Yaskawa INFORM job: OK_R2_O48(150,-90)AWOK.JBI

/JOB
//NAME OK_R2_O48(150,-90)AWOK
///FOLDERNAME X4
//POS
///NPOS 93,93,93,5,0,0
///TOOL 0
///POSTYPE PULSE
///PULSE
C00000=7128,-162535,-102538,14833,-6408,52690
C00001=-104208,-118770,-74284,45981,33291,-26248
C00002=-127942,-89719,-58931,35307,42397,-46473
C00003=-123853,-84206,-54688,32906,40963,-44702
C00004=-120909,-81305,-52666,30982,40073,-43338
C00005=-120909,-80580,-51168,31322,39602,-43537
C00006=-120933,-81321,-52095,31218,39773,-43479
C00007=-120933,-81321,-52095,31218,39773,-43479
C00008=-118429,-81278,-52077,29602,38889,-42349
C00009=-119470,-83685,-55381,29802,39949,-42541
C00010=-120965,-86018,-57149,30812,40385,-43243
C00011=-124957,-91780,-61448,33373,41616,-45066
C00012=-119941,-104378,-75649,664,44366,-1357
C00013=-114575,-89440,-58348,-34911,41926,46281
C00014=-118628,-83889,-54076,-32484,40527,44503
C00015=-120150,-81634,-52317,-31517,40024,43814
C00016=-120153,-79883,-49949,-31862,39544,44015
C00017=-120152,-80596,-50915,-31720,39740,43932
C00018=-120152,-80596,-50915,-31720,39740,43932
C00019=-122990,-80556,-50898,-29906,38725,42654
C00020=-120487,-84798,-55273,-31191,40066,43596
C00021=-118937,-87092,-57018,-32198,40551,44309
C00022=-106067,-91307,-60720,-38685,45933,49349
C00023=-98484,-126815,-102076,-39276,55586,49844
C00024=-116041,-74769,-88862,-24389,64621,38504
C00025=-110869,-91165,-78577,-23331,92195,43854
C00026=-124249,-90532,-74394,-23419,86323,40078
C00027=-124579,-90250,-73658,-23419,85946,40029
C00028=-124579,-89705,-72166,-23424,85359,40146
C00029=-124579,-90004,-72979,-23418,85679,40084
C00030=-124579,-90004,-72979,-23418,85679,40084
C00031=-127139,-89747,-72875,-23368,85013,39271
C00032=-124513,-91644,-75080,-23411,86111,40023
C00033=-122390,-96046,-81338,-23429,88175,40400
C00034=-118210,-97090,-84712,-23461,90782,41427
C00035=-128682,-92973,-79431,23550,91181,-43199
C00036=-121322,-93591,-77129,23613,87481,-41217
C00037=-119783,-92676,-74656,23621,86073,-40929
C00038=-119783,-92003,-72902,23631,85399,-41062
C00039=-119783,-92315,-73705,23625,85706,-41001
C00040=-117303,-92210,-73665,23606,85023,-40222
C00041=-119476,-92309,-74377,23618,86001,-40830
C00042=-123453,-92705,-79015,23614,89575,-41589
C00043=-126833,-58246,-59490,24431,96195,-34985
C00044=-121064,-58502,-56942,24348,92946,-33515
C00045=-122349,-90639,-72271,24283,86838,-35236
C00046=-120613,-91235,-73784,24290,86900,-34580
C00047=-121081,-75684,-65541,24266,89714,-34181
C00048=-121026,-92775,-72870,24282,85789,-34961
C00049=-121053,-101624,-76099,24352,83453,-35450
C00050=-121053,-101774,-76152,24354,83412,-35459
C00051=-121214,-86270,-68515,24620,98676,-32382
C00052=-121315,-89830,-69273,24565,98526,-32452
C00053=-128764,-80026,-69192,23683,105275,-33882
C00054=-134806,-66986,-70278,23625,104239,-34458
C00055=-107842,-77648,-85221,-23587,98114,40069
C00056=-119915,-70001,-63560,-27444,90659,45675
C00057=-122863,-62004,-57325,-27391,89936,44725
C00058=-125343,-108335,-78841,-26517,77272,26818
C00059=-123289,-107584,-77287,-26635,77411,27568
C00060=-123156,-76901,-64612,-27381,87009,45299
C00061=-123624,-94441,-71953,-27500,82842,46100
C00062=-123937,-107499,-76607,-27734,79312,46822
C00063=-123895,-107588,-76637,-27736,79301,46841
C00064=-124111,-102845,-74409,-27467,87071,44933
C00065=-123700,-99391,-71448,-27908,92704,43616
C00066=-123818,-102887,-72152,-27884,91453,43871
C00067=-113172,-80591,-67120,-26641,104065,45143
C00068=-103355,-56663,-86718,-43856,106110,10768
C00069=-95822,-140722,-117880,-57553,87470,-6427
C00070=-59504,-196684,-108230,-85963,76535,-42215
C00071=-126651,-173103,-98619,-107590,31890,-42335
C00072=-132485,-146292,-95297,-89338,25934,-52354
C00073=-127502,-141387,-93667,-80295,34491,-61924
C00074=-120359,-173692,-85938,-119295,41762,-37936
C00075=-112237,-170659,-84465,-112953,45862,-39581
C00076=-127507,-141456,-93682,-80333,34482,-61904
C00077=-127989,-162289,-111384,-72485,35866,-66585
C00078=-127720,-186855,-131843,-64092,39200,-71745
C00079=-127563,-185307,-132809,-61202,40726,-73506
C00080=-141972,-165441,-94982,-91935,28434,-22119
C00081=-120670,-166785,-110893,11236,47417,-7793
C00082=-120378,-170313,-84464,114311,39014,41261
C00083=-118671,-173407,-93959,109670,36018,44646
C00084=-117490,-116273,-97513,47995,52698,87558
C00085=-128335,-170190,-84462,108879,43427,42364
C00086=-120365,-173150,-86026,114896,39194,40925
C00087=-117457,-117591,-97936,48216,52395,87392
C00088=-108592,-156504,-118933,44933,39836,84216
C00089=-108710,-192099,-136125,56896,33409,77883
C00090=-110038,-135908,-122263,39784,48159,87867
C00091=-30894,-171068,-100229,56651,5883,46742
C00092=7128,-162535,-102538,14833,-6408,52690
BC00000=199595,668284,1075175
BC00001=291872,675689,1075175
BC00002=333462,679027,1075175
BC00003=333462,679027,1075175
BC00004=333462,679027,1075175
BC00005=333462,679027,1075175
BC00006=333462,679027,1075175
BC00007=333462,679027,1075175
BC00008=333462,679027,1075175
BC00009=333462,679027,1075175
BC00010=333462,679027,1075175
BC00011=333462,679027,1075175
BC00012=223299,677892,1075175
BC00013=102985,676652,1075175
BC00014=102985,676652,1075175
BC00015=102985,676652,1075175
BC00016=102985,676652,1075175
BC00017=102985,676652,1075175
BC00018=102985,676652,1075175
BC00019=102985,676652,1075175
BC00020=102985,676652,1075175
BC00021=102985,676652,1075175
BC00022=102985,676652,1075175
BC00023=102985,676652,1075175
BC00024=102985,676652,1075175
BC00025=115373,806609,1075175
BC00026=115373,806609,1075175
BC00027=115373,806609,1075175
BC00028=115373,806609,1075175
BC00029=115373,806609,1075175
BC00030=115373,806609,1075175
BC00031=115373,806609,1075175
BC00032=115373,806609,1075175
BC00033=115373,806609,1075175
BC00034=115373,806609,1075175
BC00035=324585,809621,1075175
BC00036=324585,809621,1075175
BC00037=324585,809621,1075175
BC00038=324585,809621,1075175
BC00039=324585,809621,1075175
BC00040=324585,809621,1075175
BC00041=324585,809621,1075175
BC00042=324585,809621,1075175
BC00043=328987,784971,1075168
BC00044=328987,784971,1075168
BC00045=328987,784969,1075175
BC00046=328987,784969,1075175
BC00047=328987,784971,1075168
BC00048=328987,784971,1075168
BC00049=328987,784971,1075168
BC00050=328987,784971,1075168
BC00051=328987,784971,1075168
BC00052=328987,784971,1075168
BC00053=328987,784971,1075168
BC00054=328987,784971,1075168
BC00055=116574,792346,1075173
BC00056=116574,792346,1075173
BC00057=116574,792346,1075173
BC00058=116574,792346,1075175
BC00059=116574,792346,1075175
BC00060=116574,792346,1075173
BC00061=116574,792346,1075173
BC00062=116574,792346,1075173
BC00063=116574,792346,1075173
BC00064=116574,792346,1075173
BC00065=116575,792346,1075173
BC00066=116575,792346,1075173
BC00067=116574,792346,1075173
BC00068=116574,737436,1075175
BC00069=122857,733121,993715
BC00070=135433,724483,830653
BC00071=135432,724483,830653
BC00072=135433,724483,830653
BC00073=135433,724483,830653
BC00074=127658,730199,812564
BC00075=127658,730199,812564
BC00076=135433,724483,830653
BC00077=135433,724483,830653
BC00078=135433,724483,830653
BC00079=135433,724483,830653
BC00080=160615,710357,862138
BC00081=210523,682360,924538
BC00082=303867,722052,847743
BC00083=303867,722052,847743
BC00084=303867,722052,847743
BC00085=311621,727375,828139
BC00086=311621,727375,828139
BC00087=303867,722052,847743
BC00088=303867,722052,847743
BC00089=303867,722052,847743
BC00090=276888,676778,849704
BC00091=235848,686978,996103
BC00092=199595,668284,1075175
EC00000=1330261,-556475
EC00001=1330261,-556475
EC00002=1330261,-556475
EC00003=1330261,-556475
EC00004=1330261,-556475
EC00005=1330261,-556475
EC00006=1330261,-556475
EC00007=1330261,-556475
EC00008=1330261,-556475
EC00009=1330261,-556475
EC00010=1330261,-556475
EC00011=1330261,-556475
EC00012=1330261,-556475
EC00013=1330261,-556475
EC00014=1330261,-556475
EC00015=1330261,-556475
EC00016=1330261,-556475
EC00017=1330261,-556475
EC00018=1330261,-556475
EC00019=1330261,-556475
EC00020=1330261,-556475
EC00021=1330261,-556475
EC00022=1330261,-556475
EC00023=1330261,-556475
EC00024=1330261,-556475
EC00025=1330261,-556475
EC00026=1330261,-556475
EC00027=1330261,-556475
EC00028=1330261,-556475
EC00029=1330261,-556475
EC00030=1330261,-556475
EC00031=1330261,-556475
EC00032=1330261,-556475
EC00033=1330261,-556475
EC00034=1330261,-556475
EC00035=1330261,-556475
EC00036=1330261,-556475
EC00037=1330261,-556475
EC00038=1330261,-556475
EC00039=1330261,-556475
EC00040=1330261,-556475
EC00041=1330261,-556475
EC00042=1330261,-556475
EC00043=1330260,-556475
EC00044=1330260,-556475
EC00045=1330261,-556475
EC00046=1330261,-556475
EC00047=1330260,-556475
EC00048=1330260,-556475
EC00049=1330260,-556475
EC00050=1330260,-556475
EC00051=1330260,-556475
EC00052=1330260,-556475
EC00053=1330260,-556475
EC00054=1330260,-556475
EC00055=1330261,-556475
EC00056=1330261,-556475
EC00057=1330261,-556475
EC00058=1330261,-556475
EC00059=1330261,-556475
EC00060=1330261,-556475
EC00061=1330261,-556475
EC00062=1330261,-556475
EC00063=1330261,-556475
EC00064=1330261,-556475
EC00065=1330261,-556475
EC00066=1330261,-556475
EC00067=1330261,-556475
EC00068=1330261,-556475
EC00069=1330261,-556475
EC00070=1330261,-556475
EC00071=1330261,-556475
EC00072=1330261,-556475
EC00073=1330261,-556475
EC00074=1330261,-556475
EC00075=1330261,-556475
EC00076=1330261,-556475
EC00077=1276882,-556475
EC00078=1207176,-556475
EC00079=1207176,-556475
EC00080=1330261,-556475
EC00081=1330261,-556475
EC00082=1330261,-556475
EC00083=1330261,-556475
EC00084=1330261,-556475
EC00085=1330261,-556475
EC00086=1330261,-556475
EC00087=1330261,-556475
EC00088=1270757,-556475
EC00089=1191966,-556475
EC00090=1191966,-556475
EC00091=1330261,-556475
EC00092=1330261,-556475
///POSTYPE BASE
///RECTAN
///RCONF 0,0,0,0,0,0,0,0,0,0,0,0,0,0,0,0,0,0,0,0,0,0,0,0
P00006=0.222,-3.123,-1.508,0.0000,0.0000,0.0000
P00021=-0.225,-6.128,-0.405,0.0000,0.0000,0.0000
P00022=0.222,-3.123,-1.508,0.0000,0.0000,0.0000
P00031=1.853,-0.001,-1.549,0.0000,0.0000,0.0000
P00032=1.957,0.503,-7.217,0.0000,0.0000,0.0000
//INST
///DATE 2025/02/06 10:35
///ATTR SC,RW
///GROUP1 RB1,BS1
///GROUP2 ST1
///LVARS 0,0,0,0,0,100,0,0
NOP
'OK_r2_O48(150,-90)
'Path S1531
MOVJ C00000 BC00000 VJ=100.00  +MOVJ EC00000 VJ=50.00
SFTOF3D
MOVJ C00001 BC00001 VJ=100.00  +MOVJ EC00001 VJ=50.00
MOVJ C00002 BC00002 VJ=100.00  +MOVJ EC00002 VJ=100.00
MOVL C00003 BC00003 V=400.0  +MOVJ EC00003 VJ=100.00
SMOVL C00004 BC00004 V=100.0  +MOVJ EC00004
SREFP 3 C00005 BC00005  +REFP EC00005
CALL JOB:SEARCH-R1-S13D
SET P021 P006
SFTON3D P021
SMOVL C00006 BC00006 V=100.0  +MOVJ EC00006
SMOVL C00007 BC00007 V=100.0  +MOVJ EC00007
SREFP 3 C00008 BC00008  +REFP EC00008
CALL JOB:SEARCH-R1-S13D
SET P021 P006
SFTON3D P021
SMOVL C00009 BC00009 V=100.0  +MOVJ EC00009
MOVL C00010 BC00010 V=400.0  +MOVJ EC00010 VJ=100.00
MOVL C00011 BC00011 V=1000.0  +MOVJ EC00011 VJ=100.00
'Path S1532
SFTOF3D
MOVJ C00012 BC00012 VJ=100.00  +MOVJ EC00012 VJ=10.00
MOVJ C00013 BC00013 VJ=100.00  +MOVJ EC00013 VJ=100.00
MOVL C00014 BC00014 V=333.3  +MOVJ EC00014 VJ=100.00
SMOVL C00015 BC00015 V=100.0  +MOVJ EC00015
SREFP 3 C00016 BC00016  +REFP EC00016
CALL JOB:SEARCH-R1-S13D
SET P022 P006
SFTON3D P022
SMOVL C00017 BC00017 V=100.0  +MOVJ EC00017
SMOVL C00018 BC00018 V=100.0  +MOVJ EC00018
SREFP 3 C00019 BC00019  +REFP EC00019
CALL JOB:SEARCH-R1-S13D
SET P022 P006
SFTON3D P022
SMOVL C00020 BC00020 V=100.0  +MOVJ EC00020
MOVL C00021 BC00021 V=400.0  +MOVJ EC00021 VJ=100.00
MOVL C00022 BC00022 V=1000.0  +MOVJ EC00022 VJ=100.00
MOVJ C00023 BC00023 VJ=100.00  +MOVJ EC00023 VJ=50.00
MOVJ C00024 BC00024 VJ=100.00  +MOVJ EC00024 VJ=100.00
'Path S1235
SFTOF3D
MOVJ C00025 BC00025 VJ=100.00  +MOVJ EC00025 VJ=100.00
MOVL C00026 BC00026 V=400.0  +MOVJ EC00026 VJ=100.00
SMOVL C00027 BC00027 V=100.0  +MOVJ EC00027
SREFP 3 C00028 BC00028  +REFP EC00028
CALL JOB:SEARCH-R1-S13D
SET P032 P006
SFTON3D P032
SMOVL C00029 BC00029 V=100.0  +MOVJ EC00029
SMOVL C00030 BC00030 V=100.0  +MOVJ EC00030
SREFP 3 C00031 BC00031  +REFP EC00031
CALL JOB:SEARCH-R1-S13D
SET P032 P006
SFTON3D P032
SMOVL C00032 BC00032 V=100.0  +MOVJ EC00032
MOVL C00033 BC00033 V=400.0  +MOVJ EC00033 VJ=100.00
MOVL C00034 BC00034 V=1000.0  +MOVJ EC00034 VJ=100.00
'Path S1204
SFTOF3D
MOVJ C00035 BC00035 VJ=100.00  +MOVJ EC00035 VJ=100.00
MOVL C00036 BC00036 V=400.0  +MOVJ EC00036 VJ=100.00
SMOVL C00037 BC00037 V=100.0  +MOVJ EC00037
SREFP 3 C00038 BC00038  +REFP EC00038
CALL JOB:SEARCH-R1-S13D
SET P031 P006
SFTON3D P031
SMOVL C00039 BC00039 V=100.0  +MOVJ EC00039
SREFP 3 C00040 BC00040  +REFP EC00040
CALL JOB:SEARCH-R1-S13D
SET P031 P006
SFTON3D P031
SMOVL C00041 BC00041 V=100.0  +MOVJ EC00041
MOVL C00042 BC00042 V=400.0  +MOVJ EC00042 VJ=100.00
SFTOF3D
'Path W341
SFTOF3D
SFTON3D P031
SMOVL C00043 BC00043 V=400.0  +MOVJ EC00043
SMOVL C00044 BC00044 V=400.0 PL=0  +MOVJ EC00044
SREFP 1 C00045 BC00045  +REFP EC00045
SREFP 2 C00046 BC00046  +REFP EC00046
MACRO1 MJ#(0) ARGF21
ARCON
SWVON WEV#(101)
SMOVL C00047 BC00047 V=8.3  +MOVJ EC00047
SMOVL C00048 BC00048 V=8.3  +MOVJ EC00048
SMOVL C00049 BC00049 V=8.3  +MOVJ EC00049
SMOVC C00050 BC00050 V=8.3  +MOVJ EC00050
SMOVC C00051 BC00051 V=8.3  +MOVJ EC00051
SMOVC C00052 BC00052 V=8.3  +MOVJ EC00052
ARCOF
SFTOF3D
SWVOF
SMOVL C00053 BC00053 V=250.0  +MOVJ EC00053
MOVJ C00054 BC00054 VJ=100.00  +MOVJ EC00054 VJ=100.00
MOVJ C00055 BC00055 VJ=100.00  +MOVJ EC00055 VJ=100.00
SFTOF3D
'Path W2042
SFTOF3D
SFTON3D P032
SMOVL C00056 BC00056 V=400.0  +MOVJ EC00056
SMOVL C00057 BC00057 V=166.7 PL=0  +MOVJ EC00057
SREFP 1 C00058 BC00058  +REFP EC00058
SREFP 2 C00059 BC00059  +REFP EC00059
ARCON
SWVON WEV#(101)
SMOVL C00060 BC00060 V=8.3  +MOVJ EC00060
SMOVL C00061 BC00061 V=8.3  +MOVJ EC00061
SMOVL C00062 BC00062 V=8.3  +MOVJ EC00062
SMOVC C00063 BC00063 V=8.3  +MOVJ EC00063
SMOVC C00064 BC00064 V=8.3  +MOVJ EC00064
SMOVC C00065 BC00065 V=10.0  +MOVJ EC00065
SMOVC C00066 BC00066 V=10.0  +MOVJ EC00066
ARCOF
SWVOF
SMOVL C00067 BC00067 V=400.0  +MOVJ EC00067
SFTOF3D
MOVJ C00068 BC00068 VJ=100.00  +MOVJ EC00068 VJ=100.00
MOVJ C00069 BC00069 VJ=100.00  +MOVJ EC00069 VJ=50.00
MOVJ C00070 BC00070 VJ=100.00  +MOVJ EC00070 VJ=100.00
SFTOF3D
'Path W1533
SFTOF3D
SFTON3D P022
MOVJ C00071 BC00071 VJ=100.00  +MOVJ EC00071 VJ=50.00
SMOVL C00072 BC00072 V=400.0  +MOVJ EC00072
SMOVL C00073 BC00073 V=133.3 PL=0  +MOVJ EC00073
SREFP 1 C00074 BC00074  +REFP EC00074
SREFP 2 C00075 BC00075  +REFP EC00075
ARCON
SWVON WEV#(101)
SMOVC C00076 BC00076 V=8.3  +MOVJ EC00076
SMOVC C00077 BC00077 V=8.3  +MOVJ EC00077
SMOVC C00078 BC00078 V=8.3  +MOVJ EC00078
ARCOF
SMOVL C00079 BC00079 V=400.0  +MOVJ EC00079
MOVJ C00080 BC00080 VJ=100.00  +MOVJ EC00080 VJ=100.00
SFTOF3D
MOVJ C00081 BC00081 VJ=100.00  +MOVJ EC00081 VJ=100.00
'Path W1535
SFTOF3D
SFTON3D P021
MOVJ C00082 BC00082 VJ=100.00  +MOVJ EC00082 VJ=100.00
SMOVL C00083 BC00083 V=400.0  +MOVJ EC00083
SMOVL C00084 BC00084 V=166.7 PL=0  +MOVJ EC00084
SREFP 1 C00085 BC00085  +REFP EC00085
SREFP 2 C00086 BC00086  +REFP EC00086
ARCON
SMOVC C00087 BC00087 V=8.3  +MOVJ EC00087
SWVON WEV#(101)
SMOVC C00088 BC00088 V=8.3  +MOVJ EC00088
SMOVC C00089 BC00089 V=8.3  +MOVJ EC00089
ARCOF
SWVOF
SMOVL C00090 BC00090 V=500.0  +MOVJ EC00090
SFTOF3D
MOVJ C00091 BC00091 VJ=100.00  +MOVJ EC00091 VJ=100.00
MOVJ C00092 BC00092 VJ=100.00  +MOVJ EC00092 VJ=100.00
END
